// ============================================================================
// FB_TON: 接通延时定时器
// 描述: 当IN为TRUE时, 经过PT时间后Q变为TRUE
// ============================================================================

FUNCTION_BLOCK FB_TON
VAR_INPUT
    IN  : BOOL;
    PT  : DINT;   // 预设时间(扫描周期)
END_VAR
VAR_OUTPUT
    Q   : BOOL;
    ET  : DINT;   // 已用时间(扫描周期)
END_VAR
VAR
    Counter   : DINT := 0;
    Running   : BOOL := FALSE;
END_VAR

BEGIN
    // IN为TRUE时启动定时器
    IF #IN THEN
        IF NOT #Running THEN
            #Running := TRUE;
            #Counter := 0;  // 复位计数器
        END_IF;

        // 计时逻辑
        IF #Running THEN
            #Counter := #Counter + 1;

            // 判断是否达到预设值
            IF #Counter >= #PT THEN
                #Q := TRUE;
                #ET := #PT;
                #Counter := #PT;  // 保持最大值
            ELSE
                #ET := #Counter;  // 输出当前值
            END_IF;
        END_IF;
    ELSE
        // IN为FALSE时复位
        #Q := FALSE;
        #ET := 0;
        #Counter := 0;
        #Running := FALSE;
    END_IF;

END_FUNCTION_BLOCK
